{attribute 'GeneratedUsingTerminal: EL3002-0000-0016'}
{attribute addProperty BoxType "EL3002-0000-0016"}
{attribute addProperty Description "EL3002 2Ch. Ana. Input +/-10V"}
{attribute addProperty Physics "KK"}
{attribute addProperty Id "AI_Standard_Channel_1AT %I*AI_Standard_Channel_EA9DF21E9AI_Standard_Channel_2AT %I*AI_Standard_Channel_EA9DF21E9WcStateAT %I*WcState_9091E0EB2InfoDataAT %I*InfoData_32EB74EA10"}
{attribute addProperty CRC "4288367364"}
{attribute addProperty Size "30"}
TYPE EL3002_FF9B4B04 EXTENDS EtcSlaveTerminalBase_947E5A46 :
STRUCT
	{attribute addProperty Name "AI_Standard_Channel_1"}
	AI_Standard_Channel_1 : AI_Standard_Channel_EA9DF21E;
	{attribute addProperty Name "AI_Standard_Channel_2"}
	AI_Standard_Channel_2 : AI_Standard_Channel_EA9DF21E;
	{attribute addProperty Name "WcState"}
	WcState : WcState_9091E0EB;
	{attribute addProperty Name "InfoData"}
	InfoData : InfoData_32EB74EA;
END_STRUCT
END_TYPE

(* stored: Version 1.2.0.0, ProductVersion 3.1.4024.11
   DUT EL3002_FF9B4B04: Id {579792fc-eac9-4bb2-9d41-b467779e6cdf} *)
